{attribute 'linkalways'} 
{attribute 'no_explicit_call' := 'This FB is a CLASS and must be accessed using methods or properties'}
{attribute 'enable_dynamic_creation'}
FUNCTION_BLOCK _ETcVnElementType EXTENDS EnumDatatypeBase
VAR
	localData : ETcVnElementType;
	activeData : REFERENCE TO ETcVnElementType;
	enumBaseDatatype : _DINT(localData);
END_VAR

METHOD PRIVATE AddLocalEnumeration
VAR_INPUT
	Enumeration : T_MAXSTRING;
	Value : ETcVnElementType;
END_VAR
AddEnumeration(Enumeration, Value);
END_METHOD

PROPERTY PUBLIC Address : PVOID
GET
Address := ADR(activeData);
END_GET
END_PROPERTY

METHOD PUBLIC ClearReference
VAR_INPUT
END_VAR
activeData REF= localData;
SetBaseDatatypeReference();
END_METHOD

METHOD PUBLIC Clone : I_Datatype
VAR
    pClone : POINTER TO _ETcVnElementType;
END_VAR
pClone := __NEW(_ETcVnElementType(InitialValue := Value));
Clone := pClone^;
END_METHOD

METHOD FB_init : BOOL
VAR_INPUT
	bInitRetains : BOOL; // if TRUE, the retain variables are initialized (warm start / cold start)
	bInCopyCode : BOOL;  // if TRUE, the instance afterwards gets moved into the copy code (online change)
	InitialValue : ETcVnElementType;
END_VAR
localData := InitialValue;
AddBaseDatatype(enumBaseDatatype);
ClearReference();

AddLocalEnumeration('TCVN_ET_SAME_AS_SOURCE', ETcVnElementType.TCVN_ET_SAME_AS_SOURCE);
AddLocalEnumeration('TCVN_ET_USINT', ETcVnElementType.TCVN_ET_USINT);
AddLocalEnumeration('TCVN_ET_SINT', ETcVnElementType.TCVN_ET_SINT);
AddLocalEnumeration('TCVN_ET_UINT', ETcVnElementType.TCVN_ET_UINT);
AddLocalEnumeration('TCVN_ET_INT', ETcVnElementType.TCVN_ET_INT);
AddLocalEnumeration('TCVN_ET_DINT', ETcVnElementType.TCVN_ET_DINT);
AddLocalEnumeration('TCVN_ET_REAL', ETcVnElementType.TCVN_ET_REAL);
AddLocalEnumeration('TCVN_ET_LREAL', ETcVnElementType.TCVN_ET_LREAL);
END_METHOD

PROPERTY PUBLIC Identifier : T_MAXSTRING
GET
Identifier := 'ETcVnElementType';
END_GET
END_PROPERTY

METHOD IsEnumeratorValueEqual : BOOL
VAR_INPUT
	Enumerator : I_KeyValueForwardEnumerator;
END_VAR
VAR
	storedValue : ETcVnElementType;
END_VAR
IF NOT Enumerator.TryGet(storedValue) THEN
	RETURN;
END_IF

IsEnumeratorValueEqual := storedValue = activeData;
END_METHOD

METHOD PUBLIC MakeReferenceTo
VAR_INPUT
	ReferenceTarget : REFERENCE TO ETcVnElementType;
END_VAR
activeData REF= ReferenceTarget;
SetBaseDatatypeReference();
END_METHOD

METHOD PROTECTED SetBaseDatatypeReference
VAR_INPUT
END_VAR
enumBaseDatatype.MakeReferenceTo(activeData);
END_METHOD

PROPERTY PUBLIC Size : UDINT
GET
Size := SIZEOF(activeData);
END_GET
END_PROPERTY

METHOD TryMakeReferenceTo : BOOL
VAR_INPUT
	Target : I_Datatype;
END_VAR
VAR
	targetAsEnum : I_EnumDatatype;
	pTargetData : POINTER TO ETcVnElementType;
END_VAR
IF NOT Target.TryResolveAsEnumDatatype(targetAsEnum) THEN
	RETURN;
END_IF

IF targetAsEnum.Identifier <> Identifier THEN
	RETURN;
END_IF

pTargetData := Target.Address;
activeData REF= pTargetData^;
SetBaseDatatypeReference();
TryMakeReferenceTo := TRUE;
END_METHOD

PROPERTY PUBLIC Value : ETcVnElementType
GET
Value := activeData;
END_GET
SET
activeData := Value;
END_SET
END_PROPERTY

END_FUNCTION_BLOCK

(* stored: Version 1.1.0.1, ProductVersion 3.1.4024.12
   POU _ETcVnElementType: Id {f02600d5-f9ab-4e42-87ce-9fa2b7315c9d}, SpecialFunc None
   Folder Constructor: Id {5c68abab-8652-42fe-b141-a36eec4b55a5}
   Folder Private: Id {6be022b2-a358-415d-ad94-796eb63f5cf3}
   Folder Protected: Id {35797a4d-ac4c-4973-8448-8dfeb0ffe3f1}
   Method AddLocalEnumeration: Id {872e222b-9da5-4631-959e-c0b8e81936d0}
   Property Address: Id {55868eec-8273-48a0-af68-d869c3db1eec}
   Get Get: Id {4c3fb2fe-cf77-4bbc-af01-2b7cb5625019}
   Method ClearReference: Id {b6168bc6-93c5-4b71-b132-8cec86e7d5c8}
   Method Clone: Id {6970dd9a-ec2f-4dff-b339-9af177537c7c}
   Method FB_init: Id {c8d39a47-57a8-4387-973e-2b01ad39013f}
   Property Identifier: Id {ac8c15e1-3451-4332-8ae3-fbf2992d09b0}
   Get Get: Id {4a81d617-29d5-4593-a29f-75a6950695da}
   Method IsEnumeratorValueEqual: Id {036e777e-041b-4bba-8bbe-187939649ac7}
   Method MakeReferenceTo: Id {760d2d97-11ad-4488-b4c3-7c8195b177cd}
   Method SetBaseDatatypeReference: Id {862c7560-84e8-4872-a624-439845ebd93b}
   Property Size: Id {f013cc14-84d1-429d-ac22-f674528cd784}
   Get Get: Id {12900cd9-790b-4755-9473-44ee2a6ab5ed}
   Method TryMakeReferenceTo: Id {3ffea9cf-f2ef-4537-bd14-4af5fb0a15fe}
   Property Value: Id {724ec425-d8b5-4d55-bfd5-007df4eef270}
   Get Get: Id {6835325d-7d23-4871-8ca3-549ee1a7ce79}
   Set Set: Id {b4a01a29-bdc4-45f8-963f-72576fd02409} *)
